Universal Robots PolyScope program: xmlrpc_deteccion_fresas_v2.urp

Program xmlrpc_deteccion_fresas_v2 (installation=default directory=/programs/usbdisk createdIn=5.17.0 lastSavedIn=5.21.3 robotSerialNumber=20185300103)
Calibrated DH parameters: a=[-0.00011, -0.177742, -0.140941, 0.000115, -0.000132, 0]; d=[0.151657, 34.818115, -45.396006, 10.707357, 0.085307, 0.091775]; alpha=[1.570734, 0.004798, -0.015068, 1.570708, -1.571204, 0]; deltaTheta=[0, 0.754463, 0.092237, -0.846764, -0.000014, 0]
InitVariablesNode
BeforeStart
  Folder Configuracion XMLRPC
    'Configuración del XMLRPC'
    camera := rpc_factory("xmlrpc","http://192.168.23.107:50000")
  Folder Inicializacipn variables
    'Configuracion offset para el pre_pick'
    z := 0.03
    offset := p[0,0,z,0,0,0]
    'Variable para ver si se detecta dos veces el mismo pto'
    next_pose_aux := p[0,0,0,0,0,0]
  Folder Centro coord camara
    'Punto de referencia de la camara (centro de coordenadas camara)'
    MoveJ speed 60 deg/s, acceleration 80 deg/s^2 (useActiveTCP=true optimoveEnabled=false optiMoveSpeed=0.3 optiMoveAcceleration=0.09) feature=Joint_6_name
      Waypoint reference_p: TCP in base x=-184.324 y=315.895 z=51.886 mm, rx=1.3563 ry=2.8337 rz=0 rad; joints [-218.985, -126.88, -111.555, -31.537, 89.124, -78.258] deg; TCP offset x=0 y=0 z=20 mm, rx=0 ry=0 rz=0 rad; feature pose in base x=-201.494 y=311.576 z=68.423 mm, rx=-0.9117 ry=-1.9163 rz=-0.0074 rad
    referencep_var := reference_p
Robot Program (runOnlyOnce=false)
  Folder Home
    'Home: Punto inicial para posterior recogida de deteccion'
    MoveJ speed 60 deg/s, acceleration 80 deg/s^2 (useActiveTCP=true optimoveEnabled=false optiMoveSpeed=0.3 optiMoveAcceleration=0.09) feature=Joint_6_name
      Waypoint Casa: TCP in base x=-78.238 y=201.293 z=163.745 mm, rx=1.3345 ry=2.8256 rz=-0.0239 rad; joints [-212.856, -66.092, -140.54, -64.401, 89.697, -72.072] deg; TCP offset x=0 y=0 z=20 mm, rx=0 ry=0 rz=0 rad
  Folder Comunicacion camara
    'Obtencion de datos de la camara'
    next_pose := camera.get_next_pose()
    'Se hace el cambio de unidades mm a m'
    next_pose_list := p[next_pose[0]/1000,next_pose[1]/1000,0,0,0,0]
    'Trasformada entre el robot y las coordenadas obtenidas'
    target := pose_trans(reference_p,next_pose_list)
    target := p[target[0],target[1],target[2],0,0,0]
  Folder Movimiento UR
    If next_pose_list[0]≟0  and next_pose_list[1]≟0
      Folder NO_Deteccion
        MoveJ speed 60 deg/s, acceleration 80 deg/s^2 (useActiveTCP=true optimoveEnabled=false optiMoveSpeed=0.3 optiMoveAcceleration=0.09) feature=Joint_6_name
          Waypoint Casa: TCP in base x=-78.238 y=201.293 z=163.745 mm, rx=1.3345 ry=2.8256 rz=-0.0239 rad; joints [-212.856, -66.092, -140.54, -64.401, 89.697, -72.072] deg; TCP offset x=0 y=0 z=20 mm, rx=0 ry=0 rz=0 rad
    Else 
      Folder Deteccion_OK
        If next_pose_aux ≠ next_pose_list
          'Hay detecciones que recoger'
          'Posicion previa a la recogida'
          pre_pick := pose_trans(target, offset)
          pre_pick := p[pre_pick[0],pre_pick[1],pre_pick[2],referencep_var[3],referencep_var[4],referencep_var[5]]
          MoveL speed 250 mm/s, acceleration 1200 mm/s^2 (useActiveTCP=true optimoveEnabled=false optiMoveSpeed=0.3 optiMoveAcceleration=0.09) feature=Base
            Waypoint Variable (Variable): variable=pre_pick
          'Variable aux para comparar listas '
          next_pose_aux := p[next_pose_list[0],next_pose_list[1],next_pose_list[2],0,0,0]
        Else 
          'No hay detecciones que recoger'
          MoveJ speed 60 deg/s, acceleration 80 deg/s^2 (useActiveTCP=true optimoveEnabled=false optiMoveSpeed=0.3 optiMoveAcceleration=0.09) feature=Joint_6_name
            Waypoint Casa: TCP in base x=-78.238 y=201.293 z=163.745 mm, rx=1.3345 ry=2.8256 rz=-0.0239 rad; joints [-212.856, -66.092, -140.54, -64.401, 89.697, -72.072] deg
  Wait Sleep waitTime=1
